TYPE ST_FSoE_10Byte :
STRUCT
	CMD		: BYTE;
	SafeData1 	: WORD;
	CRC1		: WORD;
	SafeData2 	: WORD;
	CRC2		: WORD;
	SafeData3 	: WORD;
	CRC3		: WORD;
	SafeData4 	: WORD;
	CRC4		: WORD;
	SafeData5 	: WORD;
	CRC5		: WORD;
	ConnID		: WORD;
END_STRUCT
END_TYPE

(* stored: Version 1.1.0.1, ProductVersion 3.1.4024.5
   DUT ST_FSoE_10Byte: Id {f2de064b-87d9-4d10-9f08-466d4bbd3cb3} *)
